// LS Electric XG5000 project: 최종 plc 프레임_변경안
// PLC LSPLC
// module base 0 slot 0: 입출력 모듈:XBC-DR32H (DC 24V 입력, 릴레이 출력 32점)

PROGRAM NewProgram (task: 스캔 프로그램)

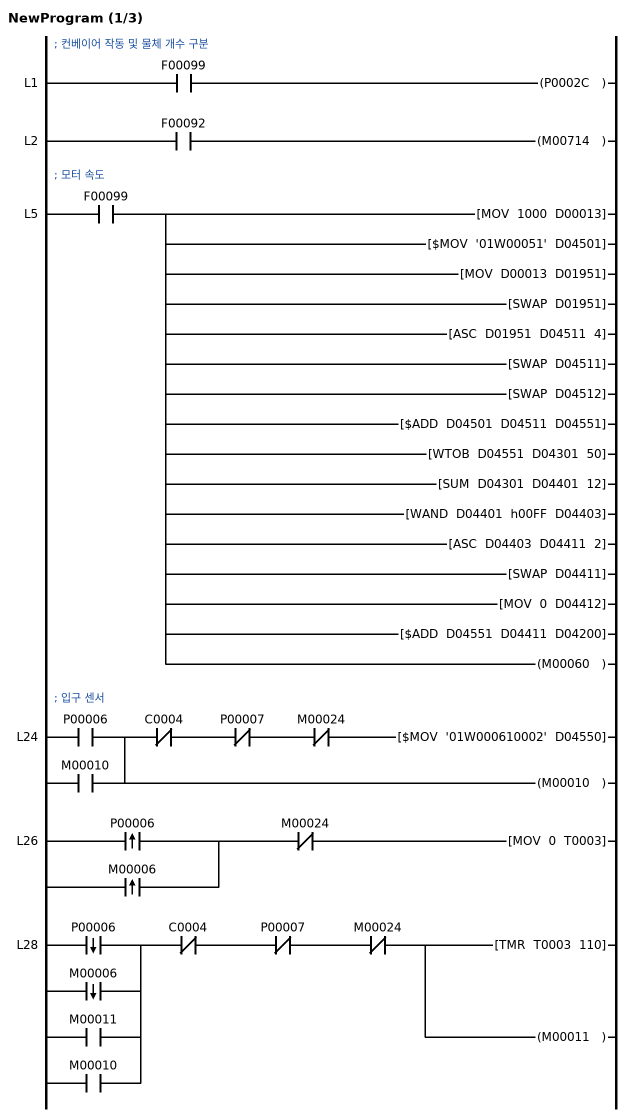
// 컨베이어 작동 및 물체 개수 구분
; L1
LOAD      F00099
OUT       P0002C
; L2
LOAD      F00092
OUT       M00714
// 모터 속도
; L5
LOAD      F00099
MOV       1000 D00013
$MOV      '01W00051' D04501
MOV       D00013 D01951
SWAP      D01951
ASC       D01951 D04511 4
SWAP      D04511
SWAP      D04512
$ADD      D04501 D04511 D04551
WTOB      D04551 D04301 50
SUM       D04301 D04401 12
WAND      D04401 h00FF D04403
ASC       D04403 D04411 2
SWAP      D04411
MOV       0 D04412
$ADD      D04551 D04411 D04200
OUT       M00060
// 입구 센서
; L24
LOAD      P00006
OR        M00010
MPUSH
AND NOT   C0004
AND NOT   P00007
AND NOT   M00024
$MOV      '01W000610002' D04550
MPOP
OUT       M00010
; L26
LOADP     P00006
ORP       M00006
AND NOT   M00024
MOV       0 T0003
; L28
LOADN     P00006
ORN       M00006
OR        M00011
OR        M00010
AND NOT   C0004
AND NOT   P00007
AND NOT   M00024
TMR       T0003 110
OUT       M00011

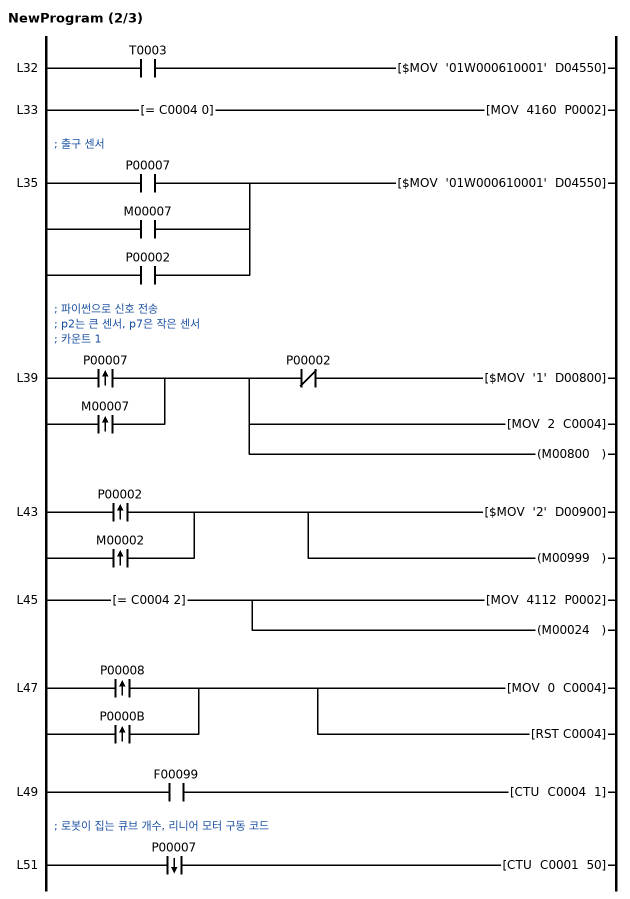
; L32
LOAD      T0003
$MOV      '01W000610001' D04550
; L33
LOAD=     C0004 0
MOV       4160 P0002
// 출구 센서
; L35
LOAD      P00007
OR        M00007
OR        P00002
$MOV      '01W000610001' D04550
; L39
LOADP     P00007
ORP       M00007
MPUSH
AND NOT   P00002
$MOV      '1' D00800
MPOP
MOV       2 C0004
OUT       M00800
// output comment: 파이썬으로 신호 전송 p2는 큰 센서, p7은 작은 센서
// output comment: 카운트 1
; L43
LOADP     P00002
ORP       M00002
$MOV      '2' D00900
OUT       M00999
; L45
LOAD=     C0004 2
MOV       4112 P0002
OUT       M00024
; L47
LOADP     P00008
ORP       P0000B
MOV       0 C0004
RST       C0004
; L49
LOAD      F00099
CTU       C0004 1
// 로봇이 집는 큐브 개수, 리니어 모터 구동 코드
; L51
LOADN     P00007
CTU       C0001 50

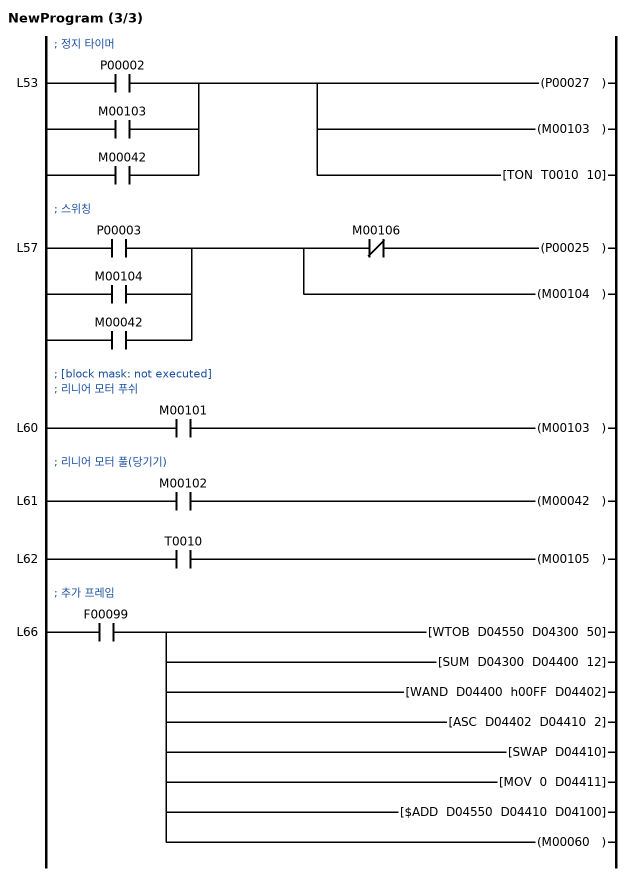
; L53
LOAD      P00002
OR        M00103
OR        M00042
OUT       P00027
OUT       M00103
TON       T0010 10
// output comment: 정지 타이머
; L57
LOAD      P00003
OR        M00104
OR        M00042
MPUSH
AND NOT   M00106
OUT       P00025
MPOP
OUT       M00104
// output comment: 스위칭
; L60 (block mask: not executed)
LOAD      M00101
OUT       M00103
// output comment: 리니어 모터 푸쉬
; L61
LOAD      M00102
OUT       M00042
// output comment: 리니어 모터 풀(당기기)
; L62
LOAD      T0010
OUT       M00105
// 추가 프레임
; L66
LOAD      F00099
WTOB      D04550 D04300 50
SUM       D04300 D04400 12
WAND      D04400 h00FF D04402
ASC       D04402 D04410 2
SWAP      D04410
MOV       0 D04411
$ADD      D04550 D04410 D04100
OUT       M00060
// 파이썬 to PLC